{region '#Template'}
	{attribute 'Version' := '5.0.0.0'}
	{attribute 'Tags' := '"LCID": "1031", "Text": "Universal, Analog, Aggregate"'}
	{attribute 'Tags' := '"LCID": "1033", "Text": "Universal, Analog, Aggregate"'}
	{attribute 'Using' := '"Type": "Template", "URI": "EC_ID"'}
	{attribute 'Using' := '"Type": "Template", "URI": "BA2_Param"'}
	{attribute 'Description' := '"LCID": "1031", "Text": "Aktor analog"'}
	{attribute 'Description' := '"LCID": "1033", "Text": "Actuator analog"'}
{endregion}
FUNCTION_BLOCK FB_BA_ActuatorMdlt EXTENDS FB_BA_View
VAR_INPUT
	stCmd					: ST_BA_Mdlt;	
	fValPgm					: REAL;
END_VAR
VAR_OUTPUT
	fMdlt					: REAL;
	bDst					: BOOL;
	eActivePrio				: E_BA_Priority;
END_VAR
VAR_INPUT CONSTANT PERSISTENT
	{attribute 'parameterCategory' := 'Behaviour'}
	fMinModulation 				: REAL := 20;
	{attribute 'parameterCategory' := 'Behaviour'}
	fMaxModulation 				: REAL := 100;
END_VAR
VAR_INPUT CONSTANT
	Mdlt					: FB_BA_AO_Raw;
	PlantLock				: FB_BA_PlantLock;	
END_VAR
VAR
	bPrioSfty					: BOOL;
	bPrioCrit					: BOOL;	
	
	PrioSwiVal					: FB_BA_PrioSwi_UDI04;	
	MuxMdlt						: FB_BA_MMUX_R04;
END_VAR

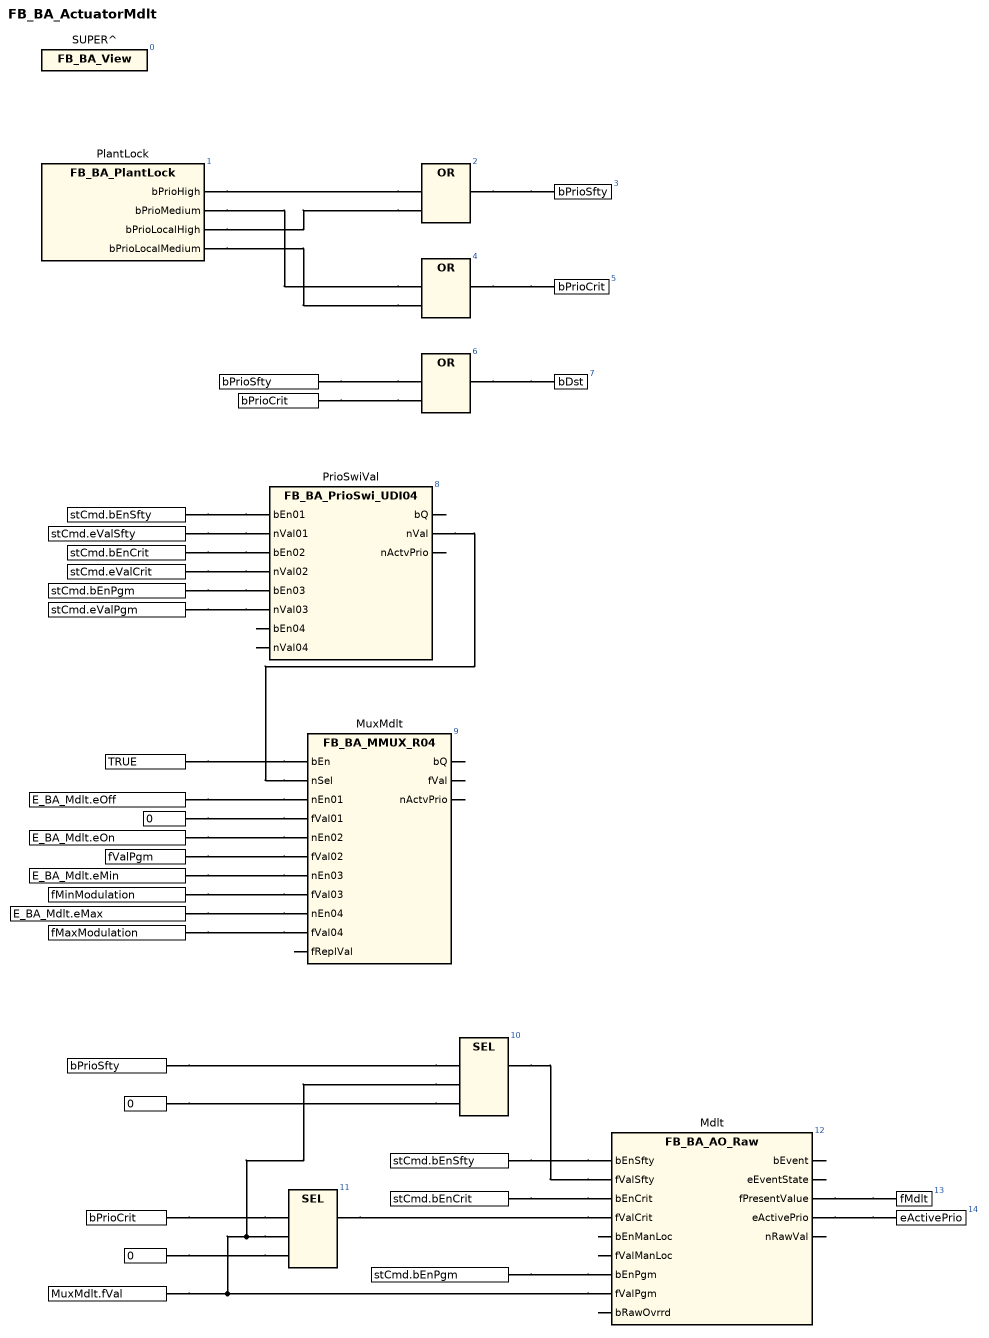
SUPER^(); // FB_BA_View
PlantLock(); // FB_BA_PlantLock
bPrioSfty := PlantLock.bPrioHigh OR PlantLock.bPrioLocalHigh;
bPrioCrit := PlantLock.bPrioMedium OR PlantLock.bPrioLocalMedium;
bDst := bPrioSfty OR bPrioCrit;
PrioSwiVal(
    bEn01 := stCmd.bEnSfty,
    nVal01 := stCmd.eValSfty,
    bEn02 := stCmd.bEnCrit,
    nVal02 := stCmd.eValCrit,
    bEn03 := stCmd.bEnPgm,
    nVal03 := stCmd.eValPgm); // FB_BA_PrioSwi_UDI04
MuxMdlt(
    bEn := TRUE,
    nSel := PrioSwiVal.nVal,
    nEn01 := E_BA_Mdlt.eOff,
    fVal01 := 0,
    nEn02 := E_BA_Mdlt.eOn,
    fVal02 := fValPgm,
    nEn03 := E_BA_Mdlt.eMin,
    fVal03 := fMinModulation,
    nEn04 := E_BA_Mdlt.eMax,
    fVal04 := fMaxModulation); // FB_BA_MMUX_R04
Mdlt(
    bEnSfty := stCmd.bEnSfty,
    fValSfty := SEL(bPrioSfty, MuxMdlt.fVal, 0),
    bEnCrit := stCmd.bEnCrit,
    fValCrit := SEL(bPrioCrit, MuxMdlt.fVal, 0),
    bEnPgm := stCmd.bEnPgm,
    fValPgm := MuxMdlt.fVal); // FB_BA_AO_Raw
fMdlt := Mdlt.fPresentValue;
eActivePrio := Mdlt.eActivePrio;

METHOD FB_init : BOOL
VAR_INPUT
	bInitRetains : BOOL; // if TRUE, the retain variables are initialized (warm start / cold start)
	bInCopyCode : BOOL;  // if TRUE, the instance afterwards gets moved into the copy code (online change)
END_VAR
PlantLock.Parent				:= THIS^;		

Mdlt.iParent					:= THIS^;
Mdlt.iLabel						:= LblFun_ControlSignal;
Mdlt.eUnit						:= E_BA_Unit.eOther_Percent;
Mdlt.fResolution 				:= 0.003051851;
Mdlt.fScaleOffset 				:= 0;
Mdlt.fCOVIncrement				:= BA2_Param.fDefCOVIncrement;
Mdlt.bEnManualRm				:= FALSE;	//	Priority  8	
Mdlt.fValManualRm				:= 0.0;		//	Priority  8
Mdlt.nEventClassID				:= EC_ID.NC80;
Mdlt.stTimeDelay.nToNormal		:= BA2_Param.nDefTimeDelay_ToNormal;
Mdlt.stTimeDelay.nToAbnormal	:= BA2_Param.nDefTimeDelay_ToAbnormal;
Mdlt.stHighLimit.bEnable		:= FALSE;
Mdlt.stHighLimit.fValue			:= 0.0;		
Mdlt.stLowLimit.bEnable			:= FALSE;
Mdlt.stLowLimit.fValue			:= 0.0;
Mdlt.fLimitDeadband 			:= BA2_Param.fDefLimitDeadband;
Mdlt.aEventTransitionText[1]	:= txtEvent_Disturb;
Mdlt.aEventTransitionText[2]	:= txtEvent_None;
Mdlt.aEventTransitionText[3]	:= txtEvent_Normal;
Mdlt.bEventDetectionEnable		:= FALSE;
Mdlt.eEnPlantLock				:= E_BA_LockPriority.eNoLock;
END_METHOD

END_FUNCTION_BLOCK

(* stored: Version 1.1.0.1, ProductVersion 3.1.4024.12
   POU FB_BA_ActuatorMdlt: Id {709fada2-7adf-415d-a5a1-846394d4338d}, SpecialFunc None
   Method FB_init: Id {32ea9b0f-cff9-4a1d-80e2-c9d5d47f2bdd} *)
